TYPE SafetyDomeAccessIOStatuses :
STRUCT
	///Is the I/O in a healthy state?
	healthStatus: HealthStatus;
END_STRUCT
END_TYPE

(* stored: Version 1.1.0.1, ProductVersion 3.1.4019.2
   DUT SafetyDomeAccessIOStatuses: Id {fab5e526-6b77-4191-89dc-3e9ca5db7168} *)
